(* IEC 61131-3 sources: repolevel_ST_code_completion/extract_code/GreatExampleOfAdvantages/FUN, 13 files *)

(* ---- GroundFloor.st ---- *)
FUNCTION_BLOCK GroundFloor
VAR_INPUT
END_VAR
VAR_OUTPUT
END_VAR
VAR
	LivingRoom:LivingRoom;
	GuestBath:GuestBathGroundFloor;
END_VAR

LivingRoom();
GuestBath();

(* ---- GuestBathGroundFloor.st ---- *)
FUNCTION_BLOCK GuestBathGroundFloor
VAR_INPUT
END_VAR
VAR_OUTPUT
END_VAR

VAR
	Lamp1:LampBase;

	ligthButton1: BOOL;

	Lamp1Out: BOOL;

	Temperature:TemperatureBase;

	//gernerates a sin as temperature
	Temp:OSCAT_BASIC.GEN_SIN;
	//MQTT
END_VAR

Lamp1(SwitchIn:= ligthButton1, LampOut=> Lamp1Out);

Temp(
	PT:= T#20S,
	AM:= 1.5,
	OS:= 20.0,
	DL:= 0.0);

Temperature(tempIn:= Temp.Out);

(* ---- Home.st ---- *)
FUNCTION_BLOCK Home
VAR_INPUT
END_VAR
VAR_OUTPUT
END_VAR
VAR
	GroundFloor:GroundFloor;
	TopFloor:TopFloor;
END_VAR

GroundFloor();
TopFloor();

(* ---- LampBase.st ---- *)
FUNCTION_BLOCK LampBase EXTENDS TopicsBase IMPLEMENTS MQTT.MQTT_SUBSCRIBE_CALLBACK
VAR_INPUT
	(*toggels lamp, sends publish*)
	SwitchIn: BOOL;

END_VAR
VAR_OUTPUT
	LampOut: BOOL;

END_VAR
VAR
	MyInit: BOOL;
	SendState:MQTT.MQTTState;
	SwitchTrigger:R_TRIG;
END_VAR

IF NOT MyInit THEN
	MyInit := TRUE;
	SUPER^();
	//this is for transmitting the lamp state
	(*SendState.Init(
	State:= ADR(LampOut),
	Topic:= ADR(MyTopicSend),
	StateName:= ADR(''),
	StateValueOn:= ADR('Lamp switched On'),
	StateValueOff:= ADR('Lamp switched Off'),
	MQTT_IN_OUT REF= GVL_MQTT.MQTT_IN_OUT,
	QoS:= SD_MQTT.QoS.ExactlyOnce,
	RetainMqtt:= TRUE);*)
	MyProperty.Collector.put(instance:= THIS^);
	SendState.Init(
	State:= ADR(LampOut),
	Topic:= ADR(MyTopicSend),
	StateName:= ADR(''),
	MQTT_IN_OUT:= GVL_MQTT.MQTT_IN_OUT,
	StateValueOn:= ADR('Lamp switched On'),
	StateValueOff:= ADR('Lamp switched Off'),
	QoS:= MQTT.QoS.ExactlyOnce,
	RetainMqtt:= TRUE);
END_IF

SwitchTrigger(CLK:= SwitchIn);
IF SwitchTrigger.Q THEN
	LampOut := LampOut XOR 1;
END_IF
SendState();

(* ---- LivingRoom.st ---- *)
FUNCTION_BLOCK LivingRoom
VAR_INPUT
END_VAR
VAR_OUTPUT
END_VAR
VAR
	Lamp1:LampBase;
	Lamp2:LampBase;
	Lamp3:LampBase;

	Temperature:TemperatureBase;

	ligthButton1: BOOL;
	ligthButton2: BOOL;
	ligthButton3: BOOL;

	Lamp1Out: BOOL;
	Lamp2Out: BOOL;
	Lamp3Out: BOOL;
	//some changing temp...
	Temp:OSCAT_BASIC.GEN_SIN;

END_VAR

Lamp1(SwitchIn:= ligthButton1, LampOut=> Lamp1Out);
Lamp2(SwitchIn:= ligthButton2, LampOut=> Lamp2Out);
Lamp3(SwitchIn:= ligthButton3, LampOut=> Lamp3Out);

Temp(
	PT:= T#30S,
	AM:= 2.0,
	OS:= 20.0,
	DL:= 0.0);

Temperature(tempIn:= Temp.Out);

(* ---- MainBath.st ---- *)
FUNCTION_BLOCK MainBath
VAR_INPUT
END_VAR
VAR_OUTPUT
END_VAR
VAR
	Lamp1:LampBase;
	Lamp2:LampBase;
	Lamp3:LampBase;

	Temperature:TemperatureBase;

	ligthButton1: BOOL;
	ligthButton2: BOOL;
	ligthButton3: BOOL;

	Lamp1Out: BOOL;
	Lamp2Out: BOOL;
	Lamp3Out: BOOL;
	//some changing temp...
	Temp:OSCAT_BASIC.GEN_SIN;

END_VAR

Lamp1(SwitchIn:= ligthButton1, LampOut=> Lamp1Out);
Lamp2(SwitchIn:= ligthButton2, LampOut=> Lamp2Out);
Lamp3(SwitchIn:= ligthButton3, LampOut=> Lamp3Out);

Temp(
	PT:= T#40S,
	AM:= 1.0,
	OS:= 20.0,
	DL:= 0.0);

Temperature(tempIn:= Temp.Out);

(* ---- MQTT_STUFF.st ---- *)
FUNCTION_BLOCK MQTT_STUFF
VAR_INPUT
END_VAR
VAR_OUTPUT
END_VAR
VAR
	//Client:SD_MQTT.HANDLE_MQTT;

	Subscriber:MQTT.MQTTSubscribe;
	init: BOOL;
	InstanceName:CommonTypesAndFunctions.GetInstanceName;
	SubscribeTopic:STRING(255);
	birthTopic:STRING(255);
	found:DINT;
	pt:POINTER TO STRING;
	birthMessage:MQTT.MQTTPublish;
	connectRising:R_TRIG;
	xxx:POINTER TO STRING;
END_VAR

IF NOT init THEN
	init := TRUE;
	Subscriber.SetMqttInOut(MQTT_IN_OUT:= GVL_MQTT.MQTT_IN_OUT);
	SubscribeTopic := InstanceName.GetInstanceTopic();
	birthTopic := SubscribeTopic;
	found := CommonTypesAndFunctions.find(str1:= ADR(SubscribeTopic), str2:= ADR('/'));
	found := found + 1 + CommonTypesAndFunctions.find(str1:= ADR(SubscribeTopic[found + 1]), str2:= ADR('/'));
	pt := ADR(SubscribeTopic[found  + 1]);
	pt^ := 'Receive/#';
	GVL_MQTT.MQTT_IN_OUT.ClientID := CONCAT('CodesysMqtt',TO_STRING(TICKS.GetTick(xDummy:= TRUE)));
END_IF

GVL_MQTT.MQTT_IN_OUT.clientFB(
	MQTT_IN_OUT:= GVL_MQTT.MQTT_IN_OUT,
	ENABLE:= TRUE,
	URL:= 'broker.hivemq.com:1883',
	TIMEOUT:= T#8S);

Subscriber(
	Subscribe:= TRUE,
	Topic:= ADR(SubscribeTopic),
	QoSSubscribe:= MQTT.QoS.ExactlyOnce,
	ExpectingString:= TRUE,
	Callback:= MyProperty.Collector);

connectRising(CLK:= GVL_MQTT.MQTT_IN_OUT.BROKER_CONNECTED);

	birthMessage(
	Topic:= ADR(birthTopic),
	PayloadString:= ADR('born'),
	PublishAsString:= TRUE,
	QoSIn:= MQTT.QoS.ExactlyOnce ,
	MRetain:= FALSE,
	send:= connectRising.Q);

(* ---- SleepingRoom.st ---- *)
FUNCTION_BLOCK SleepingRoom
VAR_INPUT
END_VAR
VAR_OUTPUT
END_VAR
VAR
	Lamp1:LampBase;

	ligthButton1: BOOL;

	Lamp1Out: BOOL;

	Temperature:TemperatureBase;

	//gernerates a sin as temperature
	Temp:OSCAT_BASIC.GEN_SIN;
END_VAR

Lamp1(SwitchIn:= ligthButton1, LampOut=> Lamp1Out);

Temp(
	PT:= T#60S,
	AM:= 1.5,
	OS:= 15.0,
	DL:= 0.0);

Temperature(tempIn:= Temp.Out);

(* ---- TemperatureBase.st ---- *)
(*this fb creats all topics an handles send and receive*)
FUNCTION_BLOCK TemperatureBase EXTENDS TopicsBase IMPLEMENTS MQTT.MQTT_SUBSCRIBE_CALLBACK
VAR_INPUT
	tempIn:REAL;
END_VAR
VAR_OUTPUT
END_VAR

VAR
	MyInit: BOOL;
	SendTemp:MQTT.MQTTValue;
	delimiter:BYTE;
	startValue:CommonTypesAndFunctions.ALL_TYPES_UNION;
	SetPoint:MQTT.ReceiveValue;
	SendPointer:CommonTypesAndFunctions.ALL_TYPES_UNION_POINTER;

END_VAR

IF NOT MyInit THEN
	MyInit := TRUE;
	SUPER^();
	SendPointer.POINTER_TO_REAL_T := ADR(tempIn);
	//prepare sending of acually temp
	SendTemp.Init(
	Topic:= ADR(MyTopicSend),
	ValueName:= ADR(''),
	ValuePointer:= SendPointer,
	ValueType:= IBaseLibrary.TYPE_REAL,
	ValueDiff:= 1,
	MQTT_IN_OUT:= GVL_MQTT.MQTT_IN_OUT,
	DecimalPlace:= 1,
	QoS:= MQTT.QoS.ExactlyOnce,
	RetainMqtt:= TRUE,
	MinTime:= T#5S);
	//init receive of temp setpoint
	SetPoint.initAsFindTopicAndPayload(
	splitChar:= ':',
	compStringTopic:= ADR(MyTopicReceive),
	compStringpayload:= ADR('Set'),
	ValueTyp:= CommonTypesAndFunctions.IBaseLibrary.TYPE_REAL,
	returnHit:= TRUE);

	MyProperty.Collector.put(THIS^);
	//init temp
	startValue.REAL_T := 22.0;
	SetPoint.SetOutput(value:= startValue);
END_IF

//here yust call sending of temp
SendTemp();

//here make some logic for your temp....
//the setpoint can be found in SetPoint.MQTTreceived.REAL_T

(* ---- TopFloor.st ---- *)
FUNCTION_BLOCK TopFloor
VAR_INPUT
END_VAR
VAR_OUTPUT
END_VAR
VAR
	MainBath:MainBath;
	SleepingRoom:SleepingRoom;
END_VAR

MainBath();
SleepingRoom();

(* ---- TopicsBase.st ---- *)
FUNCTION_BLOCK TopicsBase
VAR_INPUT
END_VAR
VAR_OUTPUT
END_VAR
VAR
	InstanceName:CommonTypesAndFunctions.GetInstanceName;
	MyTopicSend:STRING(255);
	MyTopicReceive:STRING(255);
	init: BOOL;
END_VAR

IF NOT init THEN
	init := TRUE;
	//MyTopic := InstanceName.GetInstanceTopic();
	MyTopicSend := InsertSendToStringTopic(in:= InstanceName.GetInstanceTopic(), TopicLevel:= 1);
	MyTopicReceive := InsertReceiveToStringTopic(in:= InstanceName.GetInstanceTopic(), TopicLevel:= 1);
END_IF

(* ---- LampBase_PublishReceived.st ---- *)
METHOD PublishReceived : BOOL
VAR_INPUT
	(*Collection of received Data*)
	Data	: MQTT.CALLBACK_DATA;
	(*toggels lamp, sends publish*)
	SwitchIn: BOOL;
END_VAR

VAR_OUTPUT
	LampOut: BOOL;

END_VAR
VAR
	MyInit: BOOL;
	SendState:MQTT.MQTTState;
	SwitchTrigger:R_TRIG;
END_VAR

//check if the packet is for me

IF CommonTypesAndFunctions.StrEquals(str1:= ADR(MyTopicReceive), str2:= Data.TopicOut) THEN
	PublishReceived := TRUE;//mark as done
	//now do the Commands
	IF CommonTypesAndFunctions.StrEquals(str1:= Data.PayloadString, str2:= ADR('Switch Lamp On')) THEN
		LampOut := TRUE;
	END_IF
	IF CommonTypesAndFunctions.StrEquals(str1:= Data.PayloadString, str2:= ADR('Switch Lamp Off')) THEN
		LampOut := FALSE;
	END_IF
END_IF

(* ---- TemperatureBase_PublishReceived.st ---- *)
METHOD PublishReceived : BOOL
VAR_INPUT
	(*Collection of received Data*)
	Data	: MQTT.CALLBACK_DATA;
	tempIn:REAL;
END_VAR
VAR_OUTPUT
END_VAR
VAR
	MyInit: BOOL;
	SendTemp:MQTT.MQTTValue;
	delimiter:BYTE;
	startValue:CommonTypesAndFunctions.ALL_TYPES_UNION;
	SetPoint:MQTT.ReceiveValue;
	SendPointer:CommonTypesAndFunctions.ALL_TYPES_UNION_POINTER;

END_VAR

//check if the packet is for me

PublishReceived := SetPoint.PublishReceived(Data:= Data);
